// TwinCAT 3 PLC project PLC
// ProgramVersion: 3.1.4024.0
// libraries:
//   EfficientIO Communicator, * (EfficientIO)
//   EfficientIO ModbusTCP, * (EfficientIO)
//   Lynus Persistent Data V1, * (Lynus AG)
//   Lynus Standards, * (Lynus AG)
//   Tc2_MBus, * (Beckhoff Automation GmbH)
//   Tc2_ModbusSrv, * (Beckhoff Automation GmbH)
//   Tc2_Standard, * (Beckhoff Automation GmbH)
//   Tc2_System, * (Beckhoff Automation GmbH)
//   Tc2_Utilities, * (Beckhoff Automation GmbH)
//   Tc3_IotBase, * (Beckhoff Automation GmbH)
//   Tc3_JsonXml, * (Beckhoff Automation GmbH)
//   Tc3_Module, * (Beckhoff Automation GmbH)
// project tree:
//   / FastTask.TcTTO, MiddleTask.TcTTO, SlowTask.TcTTO
//   FBs/ FB_SmartMeterAdapter.TcPOU, FB_SmartMeterAdapter_Helper.TcPOU, FB_SunSpec_PV_Inverter_T.TcPOU
//   POUs/ prgComEffIO.TcPOU, prgModbus.TcPOU, prgPersistent.TcPOU, prgRWEffIO.TcPOU, prgSMA.TcPOU, prgVarEffIO.TcPOU (not stored), prgMBUS.TcPOU
//   SolarEdge/ ST_SunSpec_PV_OutData.TcDUT
//   SolarEdge_1/ E_SunSpec_PV_Error.TcDUT, E_SunSpec_PV_OperatingState.TcDUT
// real-time tasks:
//   TASK PlcTask: cycle T#10ms, priority 20, ADS port 350
//   TASK FastTask: cycle T#10ms, priority 21, ADS port 351
//   TASK MiddleTask: cycle T#10ms, priority 22, ADS port 352
//   TASK SlowTask: cycle T#10ms, priority 23, ADS port 353
// I/O:
//   DEVICE Gerät 2 (CX-BK)
//     Box 1 (CX-BK)
// variable links:
//   PLC/PLC Instance <-> Device 2 (CX-BK)/Box 1 (CX-BK)
//     FastTask Inputs/prgMBUS.stComIn/D[{0..21}] <-> Term 2 (KL6781)/Channel 1/Data In {0..21}  (22 links)
//     FastTask Inputs/prgMBUS.stComIn/Status <-> Term 2 (KL6781)/Channel 1/Status
//     FastTask Outputs/prgMBUS.stComOut/Ctrl <-> Term 2 (KL6781)/Channel 1/Ctrl
//     FastTask Outputs/prgMBUS.stComOut/D[{0..21}] <-> Term 2 (KL6781)/Channel 1/Data Out {0..21}  (22 links)

CONFIGURATION PLC
    RESOURCE PLC ON TwinCAT3
        TASK FastTask(INTERVAL := T#10ms, PRIORITY := 21);
        TASK MiddleTask(INTERVAL := T#10ms, PRIORITY := 22);
        TASK SlowTask(INTERVAL := T#10ms, PRIORITY := 23);
        PROGRAM prgRWEffIO WITH FastTask : prgRWEffIO;
        PROGRAM prgVarEffIO WITH FastTask : prgVarEffIO;
        PROGRAM prgMBUS WITH FastTask : prgMBUS;
        PROGRAM prgPersistent WITH MiddleTask : prgPersistent;
        PROGRAM prgModbus WITH MiddleTask : prgModbus;
        PROGRAM prgSMA WITH MiddleTask : prgSMA;
        PROGRAM prgComEffIO WITH SlowTask : prgComEffIO;
    END_RESOURCE
END_CONFIGURATION

// ---- SolarEdge/ST_SunSpec_PV_OutData.TcDUT
TYPE ST_SunSpec_PV_OutData :
STRUCT
	bError					: BOOL;							//True, when the Inverter has a Error
	bFunctionIsActive		: BOOL;							//Shows if the Function is active or not
	lrPowerAcInverter		: LREAL;						//Show the actual AC Power from the Inverter in kW
	eOperatingStateInverter	: E_SunSpec_PV_OperatingState;	//Shows the Operating State from the Inverter
	eErrorState				: E_SunSpec_PV_Error;			//Error state
END_STRUCT
END_TYPE

// ---- SolarEdge_1/E_SunSpec_PV_Error.TcDUT
{attribute 'qualified_only'}
{attribute 'strict'}
TYPE E_SunSpec_PV_Error :
(
	eNoError := 0,
	eModbusTCPError := 1,
	eSunSpecError := 2,
	eSunSpecTooBigValueReceived := 3
);
END_TYPE

// ---- SolarEdge_1/E_SunSpec_PV_OperatingState.TcDUT
{attribute 'qualified_only'}
{attribute 'strict'}
TYPE E_SunSpec_PV_OperatingState :
(
	eNoDataReceived := 0,
	eOff := 1,
	eSleeping := 2,
	eStartingUp := 3,
	eTrackingPowerPoint := 4,
	eForcedPowerReduction := 5,
	eShuttingDown := 6,
	eFaults := 7,
	eStandby := 8
);
END_TYPE

// ---- POUs/prgRWEffIO.TcPOU
PROGRAM prgRWEffIO
VAR
	fbRW1		: FB_ReadWrite_v2;
END_VAR


fbRW1(
	eUploadType:= 4 ,	// every 1 minutes + change 
	bBusy=> , 
	bError=> , 
	udiErrorCodeOut=> , 
	eErrorReadWrite_Out=> );

END_PROGRAM

// ---- POUs/prgMBUS.TcPOU
PROGRAM prgMBUS
VAR
	fbMBusKL6781 : FB_MBUSKL6781;
	stComIn    AT %I*	:	ST_KL6781inData22B;
	stComOut   AT %Q*	:	ST_KL6781outData22B;
	stCom				:	ST_MBUS_Communication;
	fb_Mbus_11				: 	FB_MBUS_General_Water;
	fbmbusScan	: FB_MBUS_Scan;
	m_StartScan: BOOL;
	FB_ChangeAdress : FB_MBUS_ChangeAdr;
	m_Start 			: BOOL;
	usi_Old 			: USINT;
	usi_New	 			: USINT;
	m_Start_Change		: BOOL;
	m_Disable_Change 	: BOOL;


	
END_VAR
VAR PERSISTENT
END_VAR

fbMBusKL6781(
	usiRetries:= , 
	bStart:= , 
	bDisabled:= , 
	bBusy=> , 
	bReady=> , 
	bError=> , 
	eError=> , 
	stComIn:= stComIn, 
	stComOut:= stComOut, 
	stCom:= stCom);

fb_Mbus_11(
	usiAddress:=  , 
	stSecAdr:= , 
	eBaudrate:= E_MBUS_Baudrate.eMBus_Baud2400, 
	bStart:= m_Start, 
	bSND_NKE:= , 
	bReadInit:= , 
	tMinSendTime:= T#10S , 
	bDisabled:= , 
	bBusy=> , 
	bReady=> , 
	bError=> , 
	eError=> , 
	dwIdNumber=> , 
	byStatus=> , 
	byGEN=> , 
	byCounter=> , 
	usiRecivedAdr=> , 
	eMedium=> , 
	sMan=> , 
	stVolume=> , 
	stFlow=> , 
	stCom:= stCom);

	
// only required for commissioning the water meters	
fbMBusScan(		bStart:= m_StartScan, 
				bStop:= NOT m_StartScan, 
				eBaudrate:= E_MBUS_Baudrate.eMBus_Baud2400, 
				bDisabled:= , 
				bBusy=> , 
				bReady=> , 
				bError=> , 
				eError=> , 
				usiAddress=> , 
				usiCount=> , 
				arrDevice=> , 
				stCom:= stCom);

FB_ChangeAdress(	usiAdrOld:= usi_Old, 
					usiAdrNew:= usi_New, 
					eBaudrate:= E_MBUS_Baudrate.eMBus_Baud2400, 
					bStart:= m_Start_Change, 
					bDisabled:= m_Disable_Change, 
					bBusy=> , 
					bReady=> , 
					bError=> , 
					eError=> , 
					stCom:= stCom);

END_PROGRAM

// ---- POUs/prgPersistent.TcPOU
PROGRAM prgPersistent
VAR
	fbUSV		: FB_WritePersistentData_CX81xx;
	fb_Reboot		: NT_reboot;
	m_Reboot		: BOOL:=FALSE;
END_VAR

fbUSV(
	eSaveModeData:= eUSVSaveMode.eSaveWhenPowerfail, 
	bLoadPersistentDataOk=> , 
	bPowerFailDetect=> , 
	bError=> , 
	bySaveProcess=> , 
	dwStorageLast24h=> , 
	udiErrorCode=> );
	
		
fb_Reboot(	netid := '',
			delay := 2,
			start := m_Reboot);

END_PROGRAM

// ---- POUs/prgModbus.TcPOU
PROGRAM prgModbus
VAR
	PV1 :FB_SunSpec_PV_Inverter_T;
END_VAR

PV1(
	bEnable:= , 
	sIPAdress:= , 
	byUnitID_Inverter:= , 
	stDataSunSpec=> , 
	stDataEMPower_PV=> , 
	stDataEMCounter_PV=> , 
	diNrOfEM_OUT_PV=> );

END_PROGRAM

// ---- FBs/FB_SunSpec_PV_Inverter_T.TcPOU
// {attribute 'hide_all_locals'}
FUNCTION_BLOCK FB_SunSpec_PV_Inverter_T
VAR_INPUT PERSISTENT
	bEnable						: BOOL;												//True = Function is enabled, FALSE = Function is dissabled, no new Data
	sIPAdress					: STRING(15);										//IP Adress from the Inverter
	byUnitID_Inverter			: BYTE;												//Unit ID from the Inverter (1 to 247)
END_VAR
VAR_OUTPUT
	stDataSunSpec				: ST_SunSpec_PV_OutData;							//Output structure with Data from SunSpec
	stDataEMPower_PV			: ST_ElectricMeter_Output_Power;					//Output structure with Data from Electric Meter PV (Power Data)
	stDataEMCounter_PV			: ST_ElectricMeter_Output_Counter;					//Output structure with Data from Electric Meter PV (Counter Data)
	diNrOfEM_OUT_PV				: DINT;												//Active Number from the Electric Meter for using on other functions
END_VAR
VAR
	fbElMeter					: FB_ElectricMeter;									//Electric Meter Function 
	fbNumberDevice				: FB_NumberOfDevice;								//Function block to calcualte the number of the Device
	fbConvertEnergyRegister		: FB_CV_WORD_TO_DWORD;								//Convert function
	fbMBRead_FC3				: FB_MBReadRegs;									//Modbus Read Function (FC3)
	timDelay					: TON;												//Timer for Delay between Requests
	timTimeout					: TON;												//Timer for Timeout
	timDissableFunctions		: TON;												//Timer to dissable the Function after Lynus_Standards.Constants_General.tTimeDissableLynusFunctions Days without connection to the Lynus Cloud
	timResetConnectionOnGVL		: TON;												//Timer to try reset the connection Flag on the GVL. (When somebody delete the Connection Function and make only a onlinechange)
	FPEnable					: R_TRIG;											//Internal positive Edge
	FPError_FC_3				: R_TRIG;											//Internal positive Edge
	PD_String					: FB_PersistentData_String;							//Function to save persistent data 
	stFloat						: ST_UN_FLOAT_CONVERT_DWORD_REAL;					//Convert the Float Raw Value
	arrBuffer_FC3				: ARRAY[1..125] OF WORD;							//Buffer with Data from FC3
	arrPD						: ARRAY[1..2] OF FB_PersistentData_Number;			//Function to save persistent data 
	byWaitInStep				: BYTE;												//Wait in Step before start to clean data on PLC
	iStateGVLData				: INT;												//State machine to handle the data on the GVL
	iStateModbus				: INT;												//State variable for Statemachine
	iStateModbus_CP				: INT;												//Compare State variable
	diCounterForGVL				: DINT;												//Counter to clean old data on GVL
	lrCheckValue				: LREAL;											//Internal Value to check the value before convert
	lrTemp: LREAL;
	FB_word_to_dword: FB_CV_WORD_TO_DWORD;
	x: eByteOrder;
END_VAR

//Creator : Stefan Lackner
//Company : EfficientIO
//Date : 27.09.2022
//Version : 0.0.0.1		--> not tested yet!

//With this function its possible to read out values from the SunSpec from the manufacturer SolarEdge
//This Function read out the Values from 1 SunSpec inverter
//The protocol to the Inverter is Modbus TCP
//Attention. To access the registers, an offset of 1 must always be subtracted. Register 40001 would then be on register 40000.
//The document "sunspec-implementation-technical-note.pdf" version 2.4 got used for the Modbus adress List

//NOTE for diNr.....Designation => 
//_IN = Here Data come in from other Functions or go out to other functions about the GVL
//_OUT = Here Data go out to other functions about the GVL

(*------------------------------------------------------------------------------------------General Input Part---------------------------------------------------------------------------------------------*)

//Check limitation
byUnitID_Inverter := LIMIT(1,byUnitID_Inverter,247);

(*-------------------------------------------------------------Calcualte the number of EM System---------------------------------------------------------------*)

fbNumberDevice(
	diActualNumberOfDevices:= Lynus_Standards.GVL_Energy.stNumberOfDevices.diNumberOfElectricMeters, 
	diMaxNumberOfDevices:= Constants_Energy.diMaxNumberOfElectricMeters, 
	udiCounterOnlineChange:= TwinCAT_SystemInfoVarList._AppInfo.OnlineChangeCnt, 
	bNumberIsCalculatet=> , 
	bFPNumberIsCalculatet=> , 
	bOnlineChange=> , 
	diNumberForThisDevice=> diNrOfEM_OUT_PV, 
	diNumberOfTotalDevices=> );

//Write new Numer on GVL
IF fbNumberDevice.bFPNumberIsCalculatet THEN
	Lynus_Standards.GVL_Energy.stNumberOfDevices.diNumberOfElectricMeters := fbNumberDevice.diNumberOfTotalDevices;	
END_IF 

//Delete old Number on GVL
IF fbNumberDevice.bOnlineChange THEN 
	Lynus_Standards.GVL_Energy.stNumberOfDevices.diNumberOfElectricMeters := diNrOfEM_OUT_PV;	
		iStateGVLData := 1; 
END_IF

(*-------------------------------------------------------------Service from Backend is ready and check the connection to backend for dissabel/enable Function---------------------------------------------------------------*)

//Try to reset the variable for connection on the GVL. When all is normal then the EfficientIO Mqtt connection function set this variable to true in the next cycle
//When we have no connection to the backend then after Lynus_Standards.Constants_General.tTimeDissableLynusFunctions days the Function is dissabled with all of his functionalities
timResetConnectionOnGVL(IN:= NOT timResetConnectionOnGVL.Q, PT:= T#1H, Q=> , ET=> );
IF timResetConnectionOnGVL.Q THEN 
	Lynus_Standards.GVL_Communicator.bStateConnectionToEnableFunctions := FALSE; 
END_IF
IF NOT Lynus_Standards.GVL_Communicator.bStateConnectionToEnableFunctions THEN 
	timDissableFunctions.IN := TRUE; 
ELSE 
	timDissableFunctions.IN := FALSE; 
END_IF  
timDissableFunctions(IN:= , PT:= Lynus_Standards.Constants_General.tTimeDissableLynusFunctions, Q=> , ET=> );
	
(*------------------------------------------------------------------------------------------State Machine---------------------------------------------------------------------------------------------*)
	
//Enable
FPEnable(CLK:= bEnable, Q=> );
IF FPEnable.Q AND iStateModbus = 0 THEN 
	iStateModbus := 1; 
END_IF
IF NOT bEnable OR timDissableFunctions.Q THEN 
	iStateModbus := 0; 
END_IF

//Timer for delay
timDelay(IN:= , PT:= T#100MS, Q=> , ET=> );	

//Timer for Timeout in Statemachine
IF iStateModbus = iStateModbus_CP THEN 
	timTimeout.IN := TRUE; 
ELSE 
	timTimeout.IN := FALSE; 
END_IF
IF iStateModbus = 0 THEN 
	timTimeout.IN := FALSE; 
END_IF
timTimeout(IN:= , PT:= T#20S, Q=> , ET=> );	

//Statemachine
CASE iStateModbus OF
	
	0://Init Step
		iStateModbus_CP := iStateModbus;
		timDelay.IN := FALSE;
		
		stDataSunSpec.bFunctionIsActive := FALSE;
		stDataSunSpec.eOperatingStateInverter := E_SunSpec_PV_OperatingState.eNoDataReceived;
		fbMBRead_FC3.bExecute := FALSE;
		lrCheckValue := 0;
									
	1://Read out first Registers from 40001 to 40109
		stDataSunSpec.bFunctionIsActive := TRUE;
		iStateModbus_CP := iStateModbus;
		
		fbMBRead_FC3.nQuantity := 108;
		fbMBRead_FC3.nMBAddr := 40000;  
		fbMBRead_FC3.bExecute := TRUE;
		fbMBRead_FC3.nUnitID := byUnitID_Inverter;
			
		IF fbMBRead_FC3.bBusy THEN 
			timDelay.IN := TRUE; 
		END_IF
		
		//Wait for Delay, copy Data and then next step
		IF NOT fbMBRead_FC3.bBusy AND NOT fbMBRead_FC3.bError AND timDelay.Q AND fbMBRead_FC3.nErrId=0 AND fbMBRead_FC3.cbRead<>0 THEN
			//Copy Data Current L1
			lrCheckValue := (UINT_TO_LREAL(WORD_TO_UINT(arrBuffer_FC3[73]))*EXPT(10,(WORD_TO_INT(arrBuffer_FC3[76]))));
					//fbConvertEnergyRegister(wInputValue_1:= arrBuffer_FC3[3], wInputValue_2:= arrBuffer_FC3[4], eByteOrderForConvert:= eByteOrder.eBigEndian, dwOutputValue=> );
					//stFloat.dwRawValue := fbConvertEnergyRegister.dwOutputValue;
					//lrCheckValue := stFloat.rValueFloat;	
			IF lrCheckValue >= - 3.402823E+38 AND lrCheckValue <= 3.402823E+38 THEN 
				fbElMeter.lrCurrentL1 := lrCheckValue;
			ELSE
				iStateModbus := 300;
				stDataSunSpec.eErrorState := E_SunSpec_PV_Error.eSunSpecTooBigValueReceived;		
			END_IF
			//Copy Data Current L2
			lrCheckValue := (UINT_TO_LREAL(WORD_TO_UINT(arrBuffer_FC3[74]))*EXPT(10,(WORD_TO_INT(arrBuffer_FC3[76]))));
			IF lrCheckValue >= - 3.402823E+38 AND lrCheckValue <= 3.402823E+38 THEN 
				fbElMeter.lrCurrentL2 := lrCheckValue;
			ELSE
				iStateModbus := 300;
				stDataSunSpec.eErrorState := E_SunSpec_PV_Error.eSunSpecTooBigValueReceived;		
			END_IF
			//Copy Data Current L3
			lrCheckValue := (UINT_TO_LREAL(WORD_TO_UINT(arrBuffer_FC3[75]))*EXPT(10,(WORD_TO_INT(arrBuffer_FC3[76]))));
			IF lrCheckValue >= - 3.402823E+38 AND lrCheckValue <= 3.402823E+38 THEN 
				fbElMeter.lrCurrentL3 := lrCheckValue;
			ELSE
				iStateModbus := 300;
				stDataSunSpec.eErrorState := E_SunSpec_PV_Error.eSunSpecTooBigValueReceived;		
			END_IF
			//Copy Data Voltage L1-L2
			lrCheckValue := (UINT_TO_LREAL(WORD_TO_UINT(arrBuffer_FC3[77]))*EXPT(10,(WORD_TO_INT(arrBuffer_FC3[83]))));
			IF lrCheckValue >= - 3.402823E+38 AND lrCheckValue <= 3.402823E+38 THEN 
				fbElMeter.lrVoltageL1L2 := lrCheckValue;
			ELSE
				iStateModbus := 300;
				stDataSunSpec.eErrorState := E_SunSpec_PV_Error.eSunSpecTooBigValueReceived;		
			END_IF
			//Copy Data Voltage L2-L3
			lrCheckValue := (UINT_TO_LREAL(WORD_TO_UINT(arrBuffer_FC3[78]))*EXPT(10,(WORD_TO_INT(arrBuffer_FC3[83]))));
			IF lrCheckValue >= - 3.402823E+38 AND lrCheckValue <= 3.402823E+38 THEN 
				fbElMeter.lrVoltageL2L3 := lrCheckValue;
			ELSE
				iStateModbus := 300;
				stDataSunSpec.eErrorState := E_SunSpec_PV_Error.eSunSpecTooBigValueReceived;		
			END_IF
			//Copy Data Voltage L3-L1
			lrCheckValue := (UINT_TO_LREAL(WORD_TO_UINT(arrBuffer_FC3[79]))*EXPT(10,(WORD_TO_INT(arrBuffer_FC3[83]))));
			IF lrCheckValue >= - 3.402823E+38 AND lrCheckValue <= 3.402823E+38 THEN 
				fbElMeter.lrVoltageL3L1 := lrCheckValue;
			ELSE
				iStateModbus := 300;
				stDataSunSpec.eErrorState := E_SunSpec_PV_Error.eSunSpecTooBigValueReceived;		
			END_IF
			//Copy Data Voltage L1-N
			lrCheckValue := (UINT_TO_LREAL(WORD_TO_UINT(arrBuffer_FC3[80]))*EXPT(10,(WORD_TO_INT(arrBuffer_FC3[83]))));
			IF lrCheckValue >= - 3.402823E+38 AND lrCheckValue <= 3.402823E+38 THEN 
				fbElMeter.lrVoltageL1N := lrCheckValue;
			ELSE
				iStateModbus := 300;
				stDataSunSpec.eErrorState := E_SunSpec_PV_Error.eSunSpecTooBigValueReceived;		
			END_IF
			//Copy Data Voltage L2-N
			lrCheckValue := (UINT_TO_LREAL(WORD_TO_UINT(arrBuffer_FC3[81]))*EXPT(10,(WORD_TO_INT(arrBuffer_FC3[83]))));
			IF lrCheckValue >= - 3.402823E+38 AND lrCheckValue <= 3.402823E+38 THEN 
				fbElMeter.lrVoltageL2N := lrCheckValue;
			ELSE
				iStateModbus := 300;
				stDataSunSpec.eErrorState := E_SunSpec_PV_Error.eSunSpecTooBigValueReceived;		
			END_IF
			//Copy Data Voltage L3-N
			lrCheckValue := (UINT_TO_LREAL(WORD_TO_UINT(arrBuffer_FC3[82]))*EXPT(10,(WORD_TO_INT(arrBuffer_FC3[83]))));
			IF lrCheckValue >= - 3.402823E+38 AND lrCheckValue <= 3.402823E+38 THEN 
				fbElMeter.lrVoltageL3N := lrCheckValue;
			ELSE
				iStateModbus := 300;
				stDataSunSpec.eErrorState := E_SunSpec_PV_Error.eSunSpecTooBigValueReceived;		
			END_IF
			//Copy Data AC Power
			lrCheckValue := (UINT_TO_LREAL(WORD_TO_UINT(arrBuffer_FC3[84]))*EXPT(10,(WORD_TO_INT(arrBuffer_FC3[85]))));
			IF lrCheckValue >= - 3.402823E+38 AND lrCheckValue <= 3.402823E+38 THEN 
				fbElMeter.lrPowerTotal := lrCheckValue;
			ELSE
				iStateModbus := 300;
				stDataSunSpec.eErrorState := E_SunSpec_PV_Error.eSunSpecTooBigValueReceived;		
			END_IF
			//Copy Data Frequency
			lrCheckValue := (UINT_TO_LREAL(WORD_TO_UINT(arrBuffer_FC3[86]))*EXPT(10,(WORD_TO_INT(arrBuffer_FC3[87]))));
			IF lrCheckValue >= - 3.402823E+38 AND lrCheckValue <= 3.402823E+38 THEN 
				fbElMeter.lrFrequency := lrCheckValue;
			ELSE
				iStateModbus := 300;
				stDataSunSpec.eErrorState := E_SunSpec_PV_Error.eSunSpecTooBigValueReceived;		
			END_IF			
			//Copy Data Apparent Power
			lrCheckValue := (UINT_TO_LREAL(WORD_TO_UINT(arrBuffer_FC3[88]))*EXPT(10,(WORD_TO_INT(arrBuffer_FC3[89]))));
			IF lrCheckValue >= - 3.402823E+38 AND lrCheckValue <= 3.402823E+38 THEN 
				fbElMeter.lrApparentPowerTotal := lrCheckValue;
			ELSE
				iStateModbus := 300;
				stDataSunSpec.eErrorState := E_SunSpec_PV_Error.eSunSpecTooBigValueReceived;		
			END_IF			
			//Copy Data Reactive Power
			lrCheckValue := (UINT_TO_LREAL(WORD_TO_UINT(arrBuffer_FC3[90]))*EXPT(10,(WORD_TO_INT(arrBuffer_FC3[91]))));
			IF lrCheckValue >= - 3.402823E+38 AND lrCheckValue <= 3.402823E+38 THEN 
				fbElMeter.lrReactivePowerTotal := lrCheckValue;
			ELSE
				iStateModbus := 300;
				stDataSunSpec.eErrorState := E_SunSpec_PV_Error.eSunSpecTooBigValueReceived;		
			END_IF			
			//Copy Data AC production Energy
			FB_word_to_dword(	wInputValue_1 := arrBuffer_FC3[94],
								wInputValue_2 := arrBuffer_FC3[95],
								eByteOrderForConvert := x);
			lrCheckValue := DWORD_TO_LREAL(FB_word_to_dword.dwOutputValue)* EXPT(10,(WORD_TO_INT(arrBuffer_FC3[96])));
			IF lrCheckValue >= - 3.402823E+38 AND lrCheckValue <= 3.402823E+38 THEN 
				fbElMeter.lrCounterEnergyT1_Production := lrCheckValue / 1000;
			ELSE
				iStateModbus := 300;
				stDataSunSpec.eErrorState := E_SunSpec_PV_Error.eSunSpecTooBigValueReceived;		
			END_IF			
			//Operating State	
						(*I_STATUS_OFF			1 	Off
						I_STATUS_SLEEPING		2	Sleeping (auto-shutdown) – Night mode
						I_STATUS_STARTING		3	Grid Monitoring/wake-up
						I_STATUS_MPPT			4	Inverter is ON and producing power
						I_STATUS_THROTTLED		5	Production (curtailed)
						I_STATUS_SHUTTING_DOWN	6	Shutting down
						I_STATUS_FAULT			7	Fault
						I_STATUS_STANDBY		8	Maintenance/setup*)
	
			IF 			arrBuffer_FC3[108] = 1 THEN stDataSunSpec.eOperatingStateInverter := E_Symo_PV_OperatingState.eOff;
				ELSIF 	arrBuffer_FC3[108] = 2 THEN stDataSunSpec.eOperatingStateInverter := E_Symo_PV_OperatingState.eSleeping;
				ELSIF 	arrBuffer_FC3[108] = 3 THEN stDataSunSpec.eOperatingStateInverter := E_Symo_PV_OperatingState.eStartingUp;
				ELSIF 	arrBuffer_FC3[108] = 4 THEN stDataSunSpec.eOperatingStateInverter := E_Symo_PV_OperatingState.eTrackingPowerPoint;
				ELSIF 	arrBuffer_FC3[108] = 5 THEN stDataSunSpec.eOperatingStateInverter := E_Symo_PV_OperatingState.eForcedPowerReduction;
				ELSIF 	arrBuffer_FC3[108] = 6 THEN stDataSunSpec.eOperatingStateInverter := E_Symo_PV_OperatingState.eShuttingDown;
				ELSIF 	arrBuffer_FC3[108] = 7 THEN stDataSunSpec.eOperatingStateInverter := E_Symo_PV_OperatingState.eFaults;
				ELSIF 	arrBuffer_FC3[108] = 8 THEN stDataSunSpec.eOperatingStateInverter := E_Symo_PV_OperatingState.eStandby;
				ELSE 								stDataSunSpec.eOperatingStateInverter := E_Symo_PV_OperatingState.eNoDataReceived;
			END_IF
			//Next Step
			IF iStateModbus = 1 THEN
				fbMBRead_FC3.bExecute := FALSE;
				timDelay.IN := FALSE;
				iStateModbus := 2;
				stDataSunSpec.bError := FALSE; 
				stDataSunSpec.eErrorState := E_Symo_PV_Error.eNoError;
			END_IF
		END_IF
			
		//Error from Inverter
		IF NOT fbMBRead_FC3.bBusy AND NOT fbMBRead_FC3.bError AND timDelay.Q AND stDataSunSpec.eOperatingStateInverter = E_SunSpec_PV_OperatingState.eFaults THEN
			iStateModbus := 300;
			stDataSunSpec.eErrorState := E_Symo_PV_Error.eSymo10Error;
		END_IF
	 
		//Error or Timeout
		IF FPError_FC_3.Q OR timTimeout.Q THEN
			iStateModbus := 300;
			stDataSunSpec.eErrorState := E_SunSpec_PV_Error.eModbusTCPError;
		END_IF

	2://Wait and back to 1 step
		iStateModbus_CP := iStateModbus;
		
		iStateModbus := 1;
				
	300://Error
		iStateModbus_CP := iStateModbus;
		timDelay.IN := FALSE;
		fbMBRead_FC3.bExecute := FALSE;
		stDataSunSpec.bError := TRUE;
		iStateModbus := 1;							
END_CASE

(*------------------------------------------------------------------------------------------Modbus TCP Function---------------------------------------------------------------------------------------------*)

fbMBRead_FC3(	sIPAddr:= sIPAdress, 
				nTCPPort:= 502, 
				cbLength:= SIZEOF(arrBuffer_FC3), 
				pDestAddr:= ADR(arrBuffer_FC3), 
				tTimeout:= T#10S );

FPError_FC_3(CLK:= fbMBRead_FC3.bError, Q=> );

(*----------------------------------------------------------------------------------------Electric Meter Data----------------------------------------------------------------------------------------------*)

//Error and Warning
IF timDissableFunctions.Q THEN 
	fbElMeter.bWarning := TRUE; 
	fbElMeter.iWarningCode := 0; 
ELSE 
	fbElMeter.bWarning := FALSE; 
END_IF   

IF stDataSunSpec.bError OR Lynus_Standards.GVL_Energy.stNumberOfDevices.diNumberOfElectricMeters > Constants_Energy.diMaxNumberOfElectricMeters THEN 
	fbElMeter.bError := TRUE; 
ELSE 
	fbElMeter.bError := FALSE; 
END_IF  

IF Lynus_Standards.GVL_Energy.stNumberOfDevices.diNumberOfElectricMeters > Constants_Energy.diMaxNumberOfElectricMeters THEN 
	fbElMeter.iErrorCode := 1;
ELSIF stDataSunSpec.bError THEN 
	fbElMeter.iErrorCode := 0;
END_IF  

//Read Out Data done for EM Function
IF iStateModbus <> 2 THEN 
	fbElMeter.bReadOutDataDone := TRUE; 
ELSE 
	fbElMeter.bReadOutDataDone := FALSE; 
END_IF

//Function block for meter data
fbElMeter(
	bEnable:= bEnable AND NOT timDissableFunctions.Q, 
	bError:= , 
	bEnableReadOutFunction:= FALSE, 
	bWriteWithDelay:= TRUE,
	bPowerDataInvers:= TRUE, 
	bReadOutDataDone:= ,
	iTimeReadOutInterval:= , 
	iErrorCode:= , 
	iWarningCode:= , 
	lrTotalCounterEnergy_Consumption:= 0, 
	lrTotalCounterEnergy_Production:= , 
	lrCounterEnergyT1_Consumption:= 0, 
	lrCounterEnergyT2_Consumption:= 0, 
	lrCounterEnergyT1_Production:= , 
	lrCounterEnergyT2_Production:= 0, 
	lrCurrentL1:= , 
	lrVoltageL1N:= , 
	lrVoltageL1L2:= , 
	lrPowerL1:= 0, 
	lrCurrentL2:= , 
	lrVoltageL2N:= , 
	lrVoltageL2L3:= , 
	lrPowerL2:= 0, 
	lrCurrentL3:= , 
	lrVoltageL3N:= , 
	lrVoltageL3L1:= , 
	lrPowerL3:= 0, 
	lrPowerTotal:= , 
	lrFrequency:= , 
	lrReactivePowerTotal:= , 
	lrApparentPowerTotal:= , 
	tTimDelayOutput:= T#5S, 
	stDataEMOutPower=> , 
	stDataEMOutPowerDelay=> stDataEMPower_PV, 
	stDataEMOutCounter=> ,
	stDataEMOutCounterDelay=> stDataEMCounter_PV, 
	bReadOutMeter=> );
stDataSunSpec.lrPowerAcInverter := stDataEMPower_PV.lrPowerTotal;
(*-----------------------------------------------------------Handle data to Global structure for the Electric Meter system-----------------------------------------------------------------*)

CASE iStateGVLData OF
	
	0://Init Step
		byWaitInStep := 0;
		diCounterForGVL := 1;
	
	1://Wait for 4 Steps before clean al Data on GVL
		byWaitInStep := byWaitInStep + 1;
		IF byWaitInStep >= 4 AND fbNumberDevice.bNumberIsCalculatet THEN 
			iStateGVLData := 2; 
		END_IF
		//To much Devices, back to the Init step
		IF byWaitInStep >= 4 AND NOT fbNumberDevice.bNumberIsCalculatet THEN 
			iStateGVLData := 0; 
		END_IF	
			
	2://Clear all Data in GVL
		Lynus_Standards.GVL_Energy.stDataElectricMeters[diCounterForGVL].bEnabled := FALSE;	
		Lynus_Standards.GVL_Energy.stDataElectricMeters[diCounterForGVL].byErrorWarning := 0;
		Lynus_Standards.GVL_Energy.stDataElectricMeters[diCounterForGVL].lrCounterEnergyT1_Consumption := 0;
		Lynus_Standards.GVL_Energy.stDataElectricMeters[diCounterForGVL].lrCounterEnergyT1_Production := 0;
		Lynus_Standards.GVL_Energy.stDataElectricMeters[diCounterForGVL].lrCounterEnergyT2_Consumption := 0;
		Lynus_Standards.GVL_Energy.stDataElectricMeters[diCounterForGVL].lrCounterEnergyT2_Production := 0;
		Lynus_Standards.GVL_Energy.stDataElectricMeters[diCounterForGVL].lrPower := 0;
		Lynus_Standards.GVL_Energy.stDataElectricMeters[diCounterForGVL].lrPowerConsumption := 0;
		Lynus_Standards.GVL_Energy.stDataElectricMeters[diCounterForGVL].lrPowerConsumption := 0;
		Lynus_Standards.GVL_Energy.stDataElectricMeters[diCounterForGVL].lrPowerProduction := 0;
		Lynus_Standards.GVL_Energy.stDataElectricMeters[diCounterForGVL].lrTotalCounterEnergy_Consumption := 0;
		Lynus_Standards.GVL_Energy.stDataElectricMeters[diCounterForGVL].lrTotalCounterEnergy_Production := 0;
		
		diCounterForGVL := diCounterForGVL + 1;
		diCounterForGVL := LIMIT(0,diCounterForGVL,Constants_Energy.diMaxNumberOfElectricMeters);
		//Back to the init step
		IF diCounterForGVL >= Constants_Energy.diMaxNumberOfElectricMeters THEN 
			iStateGVLData := 0; 
		END_IF
END_CASE 	 

IF diNrOfEM_OUT_PV > 0 AND fbNumberDevice.bNumberIsCalculatet THEN
	Lynus_Standards.GVL_Energy.stDataElectricMeters[diNrOfEM_OUT_PV].bEnabled := fbElMeter.stDataEMOutPower.bEnabled;
	Lynus_Standards.GVL_Energy.stDataElectricMeters[diNrOfEM_OUT_PV].byErrorWarning := fbElMeter.stDataEMOutPower.byErrorWarning;
	Lynus_Standards.GVL_Energy.stDataElectricMeters[diNrOfEM_OUT_PV].lrCounterEnergyT1_Consumption := fbElMeter.stDataEMOutCounter.lrCounterEnergyT1_Consumption;
	Lynus_Standards.GVL_Energy.stDataElectricMeters[diNrOfEM_OUT_PV].lrCounterEnergyT1_Production := fbElMeter.stDataEMOutCounter.lrCounterEnergyT1_Production;
	Lynus_Standards.GVL_Energy.stDataElectricMeters[diNrOfEM_OUT_PV].lrCounterEnergyT2_Consumption := fbElMeter.stDataEMOutCounter.lrCounterEnergyT2_Consumption;
	Lynus_Standards.GVL_Energy.stDataElectricMeters[diNrOfEM_OUT_PV].lrCounterEnergyT2_Production := fbElMeter.stDataEMOutCounter.lrCounterEnergyT2_Production;		
	Lynus_Standards.GVL_Energy.stDataElectricMeters[diNrOfEM_OUT_PV].lrPower := fbElMeter.stDataEMOutPower.lrPowerTotal;
	Lynus_Standards.GVL_Energy.stDataElectricMeters[diNrOfEM_OUT_PV].lrPowerConsumption := fbElMeter.stDataEMOutPower.lrPowerConsumption;
	Lynus_Standards.GVL_Energy.stDataElectricMeters[diNrOfEM_OUT_PV].lrPowerProduction := fbElMeter.stDataEMOutPower.lrPowerProduction;
	Lynus_Standards.GVL_Energy.stDataElectricMeters[diNrOfEM_OUT_PV].lrTotalCounterEnergy_Consumption := fbElMeter.stDataEMOutCounter.lrTotalCounterEnergy_Consumption;
	Lynus_Standards.GVL_Energy.stDataElectricMeters[diNrOfEM_OUT_PV].lrTotalCounterEnergy_Production := fbElMeter.stDataEMOutCounter.lrTotalCounterEnergy_Production;
END_IF

(*----------------------------------------------------------Save persistent data----------------------------------------------------------------*)

arrPD[1](lrValue:= BOOL_TO_LREAL(bEnable), bEventBasedActive=> );
arrPD[2](lrValue:= BYTE_TO_LREAL(byUnitID_Inverter), bEventBasedActive=> );
PD_String(sText:= sIPAdress, bEventBasedActive=> );

END_FUNCTION_BLOCK

// ---- POUs/prgSMA.TcPOU
PROGRAM prgSMA
VAR
	fbSMA : FB_SmartMeterAdapter;
	lrenergy_consumption			: LREAL;		//{#lynus.ag#()}
	lrenergy_production				: LREAL;		//{#lynus.ag#()}
	lrreactive_energy_consumption	: LREAL;		//{#lynus.ag#()}
	lrreactive_energy_production	: LREAL;		//{#lynus.ag#()}
	lrpower_consumption				: LREAL;		//{#lynus.ag#()}
	lrpower_production				: LREAL;		//{#lynus.ag#()}
	lrreactive_power_consumption	: LREAL;		//{#lynus.ag#()}
	lrreactive_power_production		: LREAL;		//{#lynus.ag#()}
	lrpower_total					: LREAL;		//{#lynus.ag#()}
END_VAR
VAR PERSISTENT
// trigger command execution
	bEnableSMA 						: BOOL;			//{#lynus.ag#()}
END_VAR

fbSMA(
	bStart:= bEnableSMA, 
	tDelayRequest:= T#10S, 
	sHostname:= '192.168.1.20', 
	bValidResult=> , 
	bBusy=> , 
	bError=> , 
	bDone=> , 
	hrErrorCode=> ,
	lrenergy_consumption => lrenergy_consumption,
	lrenergy_production => lrenergy_production,
	lrreactive_energy_consumption => lrreactive_energy_consumption,
	lrreactive_energy_production => lrreactive_energy_production,
	lrpower_consumption => lrpower_consumption,
	lrpower_production => lrpower_production,
	lrreactive_power_consumption => lrreactive_power_consumption,
	lrreactive_power_production => lrreactive_power_production,
	lrpower_total => lrpower_total );

END_PROGRAM

// ---- FBs/FB_SmartMeterAdapter.TcPOU
FUNCTION_BLOCK FB_SmartMeterAdapter
VAR_INPUT
	bStart				: BOOL;
	tDelayRequest		: TIME;		//Timer for delay before start with the next read or write Request
	sHostname			: STRING(255);		//Hostname or IP Adress from the Server
END_VAR

VAR_IN_OUT
END_VAR

VAR_OUTPUT
	bValidResult		: BOOL;							//Valid Result received from Server
    bBusy				: BOOL;							//Function is Busy
    bError				: BOOL;							//Error sucess
	bDone				: BOOL;							//True after the decoding from the received Json File
	bConnected			: BOOL;							//Connection to the Server
	lrenergy_consumption: LREAL;
	lrenergy_production: LREAL;
	lrreactive_energy_consumption: LREAL;
	lrreactive_energy_production: LREAL;
	lrpower_consumption: LREAL;
	lrpower_production: LREAL;
	lrreactive_power_consumption: LREAL;
	lrreactive_power_production: LREAL;
	lrpower_total		: LREAL;
	hrErrorCode       	: HRESULT;						//Error Result from Http Client
END_VAR

VAR
	fbClient			: FB_IotHttpClient;
	fbHttpGet			: FB_SmartMeterAdapter_Helper;
	timStartRequest		: TON;							//Timer to Start the Request
	FPStartRequest		: R_TRIG;						//Internal positive Edge
	FPDone				: R_TRIG;						//Internal positive Edge
	FNStart				: F_TRIG;						//Internal negative Edge
END_VAR

(*------------------------------------------------------------------------------------Configure HTTP Client------------------------------------------------------------------------------------------------------*)

fbClient.sHostName := sHostname;
fbClient.tConnectionTimeout := T#30S;

IF NOT fbClient.bConfigured THEN 
	fbClient.nHostPort:= 80;
	fbClient.bKeepAlive := TRUE;
	fbClient.tConnectionTimeout := T#30S;
END_IF


//Timer to start the Request
FPStartRequest(CLK:= bStart, Q=> );
	timStartRequest(IN:= fbClient.bConfigured AND bStart AND NOT timStartRequest.Q, PT:= tDelayRequest, Q=> , ET=> );
		IF ((timStartRequest.Q AND NOT bBusy) OR (FPStartRequest.Q AND NOT bBusy AND fbClient.bConfigured)) THEN fbHttpGet.bSend := TRUE; END_IF

				
//Http Get Function
fbHttpGet(
	lrenergy_consumption => lrenergy_consumption,
	lrenergy_production => lrenergy_production,
	lrreactive_energy_consumption => lrreactive_energy_consumption,
	lrreactive_energy_production => lrreactive_energy_production,
	lrpower_consumption => lrpower_consumption,
	lrpower_production => lrpower_production,
	lrreactive_power_consumption => lrreactive_power_consumption,
	lrreactive_power_production => lrreactive_power_production,
	lrpower_total => lrpower_total,
	bSend:= , 
	fbClient:= fbClient, 
	bBusy=> bBusy, 
	bError=> );


fbHttpGet.bSend := FALSE;

FPDone(CLK:= bDone, Q=> );


fbClient.Execute();

//Error
IF fbHttpGet.bError OR fbClient.bError THEN bError := TRUE; ELSE bError := FALSE; END_IF	
	hrErrorCode := fbClient.hrErrorCode;

END_FUNCTION_BLOCK

// ---- FBs/FB_SmartMeterAdapter_Helper.TcPOU
FUNCTION_BLOCK FB_SmartMeterAdapter_Helper
VAR_INPUT
	bSend				: BOOL;
END_VAR

VAR_IN_OUT
	fbClient			: FB_IotHttpClient;
END_VAR

VAR_OUTPUT
	bBusy				: BOOL;
	bError				: BOOL;
	
	lrenergy_consumption: LREAL;
	lrenergy_production: LREAL;
	lrreactive_energy_consumption: LREAL;
	lrreactive_energy_production: LREAL;
	lrpower_consumption: LREAL;
	lrpower_production: LREAL;
	lrreactive_power_consumption: LREAL;
	lrreactive_power_production: LREAL;
	lrpower_total		: LREAL;

END_VAR

VAR
	fbRequestSMA		: FB_IotHttpRequest;
	fbJson				: FB_JsonDomParser;
	nState				: UDINT;
	RisingEdge			: R_TRIG;
	timTimeout			: TON;
	tTimeOut			: TIME := T#50S;
	bGetContentResult	: BOOL;
	sContent			: STRING(2048);
	sContent2			: STRING(2048);
	
	bGetJsonResult		: BOOL;
	jsonDoc				: SJsonValue;
	jsonDocRaw			: SJsonValue;
	jsonVal				: SJsonValue;
	
	nReqCount			: UDINT;	
	nResCount			: UDINT;
	nValidResCount		: UDINT;
	nErrCount			: UDINT;
END_VAR

//Timer for Timeout
timTimeout(IN:= nState = 1 AND bBusy, PT:= tTimeOut, Q=> , ET=> );
	IF timTimeout.Q THEN 
		nState := 0;
		bBusy := FALSE;
	END_IF

RisingEdge(CLK:= bSend );
CASE nState OF
0:	
	IF RisingEdge.Q THEN 
		IF 
			fbRequestSMA.SendRequest(sUri:='/getLastData?user=FCF5C49B1AFB&password=10164987', fbClient:=fbClient, eRequestType:=ETcIotHttpRequestType.HTTP_Get, 0, 0, 0) THEN				
			nState:= 1;
			nReqCount:= nReqCount+1;
			bBusy:= TRUE;
			bError:= FALSE;
		END_IF					
	END_IF
1:
	IF NOT fbRequestSMA.bBusy THEN
		bError:= TRUE;
		IF NOT fbRequestSMA.bError THEN				 
			bGetContentResult:= fbRequestSMA.GetContent(pContent:= ADR(sContent), nContentSize:= SIZEOF(sContent), bSetNullTermination:= TRUE);
			IF fbRequestSMA.nStatusCode >= 200 AND fbRequestSMA.nStatusCode < 300 THEN
				bGetJsonResult:= FALSE;
				FindAndReplaceChar(pSrcString:=ADR(sContent), sDeleteChar:='$N', sInsertChar:='' ,pDstString:=ADR(sContent2), nDstSize:=SIZEOF(sContent2));
				jsonDoc := fbJson.ParseDocument(sContent2);
				IF jsonDoc <> 0 THEN
					bGetJsonResult:= TRUE;
					IF fbJson.HasMember(jsonDoc, 'timestamp')  THEN
						jsonVal:= fbJson.FindMember(jsonDoc, '1.8.0');
						nValidResCount:= nValidResCount+1;
						IF fbJson.IsString(jsonVal) THEN
							lrenergy_consumption := STRING_TO_LREAL(fbJson.GetString(jsonVal)) / 1000;
						END_IF
						jsonVal:= fbJson.FindMember(jsonDoc, '2.8.0');
						nValidResCount:= nValidResCount+1;
						IF fbJson.IsString(jsonVal) THEN
							lrenergy_production := STRING_TO_LREAL(fbJson.GetString(jsonVal)) / 1000;
						END_IF
						jsonVal:= fbJson.FindMember(jsonDoc, '3.8.0');
						nValidResCount:= nValidResCount+1;
						IF fbJson.IsString(jsonVal) THEN
							lrreactive_energy_consumption := STRING_TO_LREAL(fbJson.GetString(jsonVal)) / 1000;
						END_IF
						jsonVal:= fbJson.FindMember(jsonDoc, '4.8.0');
						nValidResCount:= nValidResCount+1;
						IF fbJson.IsString(jsonVal) THEN
							lrreactive_energy_production := STRING_TO_LREAL(fbJson.GetString(jsonVal)) / 1000;
						END_IF
						jsonVal:= fbJson.FindMember(jsonDoc, '1.7.0');
						nValidResCount:= nValidResCount+1;
						IF fbJson.IsString(jsonVal) THEN
							lrpower_consumption := STRING_TO_LREAL(fbJson.GetString(jsonVal)) / 1000;
						END_IF	
						jsonVal:= fbJson.FindMember(jsonDoc, '2.7.0');
						nValidResCount:= nValidResCount+1;
						IF fbJson.IsString(jsonVal) THEN
							lrpower_production := STRING_TO_LREAL(fbJson.GetString(jsonVal)) / 1000;
						END_IF
						jsonVal:= fbJson.FindMember(jsonDoc, '3.7.0');
						nValidResCount:= nValidResCount+1;
						IF fbJson.IsString(jsonVal) THEN
							lrreactive_power_consumption := STRING_TO_LREAL(fbJson.GetString(jsonVal)) / 1000;
						END_IF	
						jsonVal:= fbJson.FindMember(jsonDoc, '4.7.0');
						nValidResCount:= nValidResCount+1;
						IF fbJson.IsString(jsonVal) THEN
							lrreactive_power_production := STRING_TO_LREAL(fbJson.GetString(jsonVal)) / 1000;
						END_IF
						jsonVal:= fbJson.FindMember(jsonDoc, '16.7.0');
						nValidResCount:= nValidResCount+1;
						IF fbJson.IsString(jsonVal) THEN
							lrpower_total := STRING_TO_LREAL(fbJson.GetString(jsonVal)) / 1000;
						END_IF	
						bError:= FALSE;
						END_IF
					END_IF						
				nResCount:= nResCount+1;			
				END_IF
		END_IF
				
		nState:= 0;
		bBusy:= FALSE;
		IF bError THEN
			nErrCount:= nErrCount+1;
		END_IF
	END_IF  	
END_CASE

END_FUNCTION_BLOCK

// ---- POUs/prgComEffIO.TcPOU
PROGRAM prgComEffIO
VAR
	fbCom		: FB_MqttCommunicator;
END_VAR

fbCom(
	bConnect:= TRUE, 
	sUserName:= '38ab59b7-5528-4708-a26c-1d3a10538b8d', 					// adopt MQTT Username
	sUserPassword:= '7470194c-4de7-4b1e-b55f-48d0fd5715b4', 				// adopt MQTT Password
	eSavePositionCertificate:= eSavePositionOnPLC.ePostionHardDisk, 
	bConnected=> , 
	bError=> , 
	hrErrorCode=> , 
	eConnectionState=> , 
	eErrorMessage_Out=> );

END_PROGRAM
